TYPE ATL :
STRUCT
(*------OBLIGATORIO-------------------*)
(*Sistema PE Com*)
PE_COM:PE_COM;

(*Sistema PE *)
PE:PE;
(*-----------------------------------*)


END_STRUCT
END_TYPE

(* stored: Version 1.1.0.1, ProductVersion 3.1.4024.9
   DUT ATL: Id {e28fcb8f-75d7-40a4-b8fa-830db39a8ef1} *)
